       //----------------------------------------------------------------------
       // 1000 mbar switches (APS)
       //----------------------------------------------------------------------
       // delayed 1000 mbar furnace chamber
       //----------------------------------
       #iTime := S_ODT(   
                   T_NO:= "BM_VAC_TMR_APS_FCH",              // Timer
                   S   := "PDI".FCH_APS,                     // Start Condition
                   TV  := #DELAY_APS_FCH,                   // Time Setpoint
                   R   := NOT "PDI".FCH_APS,                 // Reset Condition
                   BI  => #BI_TMR_APS_FCH,                  // Current Time Value
                   Q   => "DV".APS_FCH_DELAYED);             // Output


       // delayed 1000 mbar gate
       //-----------------------
       #iTime := S_ODT(   
                   T_NO:= "BM_VAC_TMR_APS_GCH",            // Timer
                   S   := "PDI".GCH_APS,                   // Start Condition
                   TV  := #DELAY_APS_GCH,                 // Time Setpoint
                   R   := NOT "PDI".GCH_APS,               // Reset Condition
                   BI  => #BI_TMR_APS_GCH,                // Current Time Value
                   Q   => "DV".APS_GCH_DELAYED);           // Output

       // delayed 1000 mbar feeder
       //-------------------------
       #iTime := S_ODT(   
                   T_NO:= "BM_VAC_TMR_APS_FDR",            // Timer
                   S   := "PDI".FDR_APS,                   // Start Condition
                   TV  := #DELAY_APS_FDR,                 // Time Setpoint
                   R   := NOT "PDI".FDR_APS,               // Reset Condition
                   BI  => #BI_TMR_APS_FDR,                // Current Time Value
                   Q   => "DV".APS_FDR_DELAYED);           // Output

       // delayed 1000 mbar main filter
       //------------------------------
       #iTime := S_ODT(   
                   T_NO:= "BM_VAC_TMR_APS_FIL",            // Timer
                   S   := "PDI".FIL_APS,                   // Start Condition
                   TV  := #DELAY_APS_FIL,                 // Time Setpoint
                   R   := NOT "PDI".FIL_APS,               // Reset Condition
                   BI  => #BI_TMR_APS_FIL,                // Current Time Value
                   Q   => "DV".APS_FIL_DELAYED);           // Output

       // delayed 1000 mbar bypass filter
       //--------------------------------
       #iTime := S_ODT(   
                   T_NO:= "BM_VAC_TMR_APS_BY_FIL",            // Timer
                   S   := "PDI".FIL_2_APS,                   // Start Condition
                   TV  := #DELAY_APS_BY_FIL,                 // Time Setpoint
                   R   := NOT "PDI".FIL_2_APS,               // Reset Condition
                   BI  => #BI_TMR_APS_BY_FIL,                // Current Time Value
                   Q   => "DV".APS_BY_FIL_DELAYED);           // Output


       "LT".CGT_APS      := "DV".APS_GCH_DELAYED;
       "LT".CLF_APS      := "DV".APS_FCH_DELAYED;
       "LT".FDR_APS      := "DV".APS_FDR_DELAYED;
       "LT".FIL_APS      := "DV".APS_FIL_DELAYED;
       "LT".BY_FIL_APS   := "DV".APS_BY_FIL_DELAYED;

       //----------------------------------------------------------------------
       // Select and set output for gas flow 1+2
       //----------------------------------------------------------------------
       "P_BM_SET_GAS_FLW_MFC_1":P := "CM_INSELECT"(auto := ("APC".AUTOMATIC AND NOT "SY".CTL_GAS_FLOW_SMI) OR "DV".SI_FIL_FSH_SEQ_ON,
                                           track:= true,
                                           ac   := "AC".SET_GAS_1_FLW,
                                           kya  := "KYA".SET_GAS_1_FLW);


       "P_BM_SET_GAS_FLW_MFC_2":P := "CM_INSELECT"(auto := "APC".AUTOMATIC AND NOT "SY".CTL_GAS_FLOW_SMI,
                                           track:= true,
                                           ac   := "AC".SET_GAS_2_FLW,
                                           kya  := "KYA".SET_GAS_2_FLW);
       IF NOT "SY".SIM_ON THEN
           "DIS".ACT_GAS_1_FLW    := "P_BM_ACT_GAS_FLW_MFC_1":P;
           "DIS".ACT_GAS_2_FLW    := "P_BM_ACT_GAS_FLW_MFC_2":P;
       END_IF;

       "LT".V16_1_OPEN := ("DIS".ACT_GAS_1_FLW>0.0) AND ("PDO".V5 OR "PDO".V6);
       "LT".V16_2_OPEN := ("DIS".ACT_GAS_2_FLW>0.0) AND ("PDO".V5 OR "PDO".V6);

       //reset manual gas flow setpoint when inlet valves are not open
       //-------------------------------------------------------------
       IF NOT ("LT".V5_OPEN OR "LT".V6_OPEN)   THEN
           "KYA".SET_GAS_1_FLW   :=  0.0;
           "KYA".SET_GAS_2_FLW   :=  0.0;
       END_IF;

       //--------------------------------------------------------------------
       //Process pump P1
       //--------------------------------------------------------------------
       "CM_ITL_IO"(ADR := 1,
                 KYD_ON := ("KYD".P1_ON OR "DV".PWR_FAIL_P1_ON),
                 KYD_OFF:= "KYD".P1_OFF,
                 AUTO := "APC".AUTOMATIC OR "DV".SI_FIL_FSH_SEQ_ON,
                 DC_ON:= "DC".P1_ON,
                 CON1 := "PDI".EMO, 
                 CON2 := NOT "DV".MAIN_LINE_FAULT, 
                 CON3 := "DV".MAIN_SWITCH_ON,
                 CON4 := "PDI".P1_FLT,
                 CON5 := NOT #Flt_P1,
                 CON6 := NOT "FLT".P1_TMP_HIGH,
                 CON7 := "SysLog1",
                 CON8 := "SysLog1",
                 ITL_OUT:= "STA_ITL_CAUSE",
                 LT_OUT := "LT".P1_ON);

       //delay P1 start
       //--------------
       "PDO".P1_ON   := "SysOndelay"( DIN := "LT".P1_ON,
                               SetTime := 10,                              // setp. time
                               ActTime := #p1_on_dly,                       // act. time
                               Tick    := "SysTick100ms");                   // timebase (1s)

       #P1_IS_ON := "PDO".P1_ON AND NOT "PDI".P1_IS_ON;             //PDI.P1_IS_ON = false: pump is running; true: pump is off

       #P1_NOT_READY := "SysOndelay"( DIN := "PDO".P1_ON AND "PDI".P1_IS_ON,
                               SetTime := 3,                           // setp. time
                               ActTime := #FltTimeP1,                   // act. time
                               Tick    := "SysTick1s");                  // timebase (1s)

       IF ("PDO".P1_ON AND #P1_NOT_READY) THEN
           #Flt_P1 := true;
       END_IF;
       (*
       //motor temperature monitoring of pump P1
       //---------------------------------------
       FLT.P1_TMP_HIGH := SysOndelay(  DIN     := NOT PDI.MON_TMP_P1,
                                       SetTime := 5,                           // setp. time
                                       ActTime := tmp_flt_p1_dly,              // act. time
                                       Tick    := SysTick1s);                  // timebase (1s)
       *)
       //reset of PTC tripping devices pump 1 and pump 2
       //-----------------------------------------------
       "LT".RST_SIHI_PU  := "SysOffdelay"( DIN     := "KYD".RST_SIHI_PU,          // reset button HMI
                                       SetTime := 10,                      // setp. time
                                       ActTime := #tmp_flt_p1_dly,          // act. time
                                       Tick    := "SysTick100ms");

       "PDO".MON_TMP_P2_RES :=  "LT".RST_SIHI_PU;     //output used for both pumps - P1 and P2                                

       //Read out SPGuard
       //-------------------------------------
       #Dprd_P1_RetVal  :=  DPRD_DAT(   LADDR  :=  16#400,             //addr1024 
                                        RECORD =>  #P1_DATA); 

       "DIS".ACT_VIB_P1          := (BYTE_TO_INT(#P1_DATA[1])-48)* 1000.0 + (BYTE_TO_INT(#P1_DATA[2])-48)*100.0 + 
                                  (BYTE_TO_INT(#P1_DATA[3])-48)*10.0 + (BYTE_TO_INT(#P1_DATA[4])-48)*1.0;
       "DIS".ACT_GEAR_OIL_TMP_P1 := (BYTE_TO_INT(#P1_DATA[6])-48)*10.0 + (BYTE_TO_INT(#P1_DATA[7])-48)* 1.0;

       "FLT".P1 := #Flt_P1 OR NOT "PDI".P1_FLT;    
       "FLT".MSR_P1_VIB           := "DIS".ACT_VIB_P1 > 149.0;
       "FLT".P1_GEAR_OIL_TMP_WRN  := "DIS".ACT_GEAR_OIL_TMP_P1> 60.0;
       "FLT".P1_GEAR_OIL_TMP_ALM  := "DIS".ACT_GEAR_OIL_TMP_P1>70.0;
       "FLT".P1_SP_WRN            := "PDI".P1_WRN OR (#P1_DATA[8]=B#16#31); 

       //--------------------------------------------------------------------
       //V10 SECUVAC Ventil P1
       //--------------------------------------------------------------------
       "PDO".V10 := "PDO".P1_ON;

       //----------------------------------------------------------------------
       // V9_1 open/close : Vacuum pump 1 seal gas         
       //----------------------------------------------------------------------
       (*
       V9_1_dly_op := SysOndelay(  DIN     := PDO.P1_ON,
                                   SetTime := 10,                      // setp. time
                                   ActTime := DelayV9_1,               // act. time
                                   Tick    := SysTick1s);              // timebase (1s)
       *)                            
       //seal gas valve vacuum pump 1 - valve opened before pump starts
       //--------------------------------------------------------------
       "PDO".P1_SEAL_GAS :=  "SysOffdelay"(DIN     := "PDI".EMO AND "DV".MAIN_SWITCH_ON AND "LT".P1_ON,
                                       SetTime := 3600,                        // setp. time
                                       ActTime := #p1_seal_gas_off_dly,         // act. time
                                       Tick    := "SysTick1s");                  // timebase (1s)
       (*
       //gas ballast valve vacuum pump 1
       //-------------------------------
       PDO.P1_GAS_BAL :=       PDI.EMO 
                           AND DV.MAIN_SWITCH_ON 
                           AND PDO.P1_ON
                           AND DV.P1_GAS_BAL_ENB;
       *)
       //--------------------------------------------------------------------
       //Booster pump P2
       //--------------------------------------------------------------------
       "PDO".P2_ON := "PDO".P1_ON AND NOT "FLT".P2_TMP_HIGH;
       "PDO".P2_FU_ON := "PDO".P1_ON AND #V2_ONDELAY_OVER;

       #P2_NOT_READY := "SysOndelay"( DIN := "PDO".P2_FU_ON AND NOT "PDI".FU_P2_RDY,
                               SetTime := 5,                           // setp. time
                               ActTime := #FltTimeP2,                   // act. time
                               Tick    := "SysTick1s");                  // timebase (1s)

       IF ("PDO".P2_FU_ON AND #P2_NOT_READY) THEN
           #Flt_P2 := true;
       ELSE
           #Flt_P2 := false;
       END_IF;

       "FLT".P2 := #Flt_P2;

       "PDO".P2_FU_RES := "KYD".ALARM_ACKN AND NOT #P2_NOT_READY;   

       //motor temperature monitoring of pump P2
       //---------------------------------------
       "FLT".P2_TMP_HIGH := "SysOndelay"(  DIN     := "PDI".MON_TMP_P2,
                                       SetTime := 5,                           // setp. time
                                       ActTime := #tmp_flt_p2_dly,              // act. time
                                       Tick    := "SysTick1s");                  // timebase (1s)

       //--------------------------------------------------------------------
       //Process pump P3
       //--------------------------------------------------------------------
       #mob_fdr_p3_off_req  :=  #mob_fdr_p3_on_req AND NOT "DV".MOB_FDR_P3_ON_REQ;
       #mob_fdr_p3_on_req   :=  "DV".MOB_FDR_P3_ON_REQ;

       "CM_ITL_IO"(ADR := 2,
                 KYD_ON := ("KYD".P3_ON OR "DV".PWR_FAIL_P3_ON OR "DV".MOB_FDR_P3_ON_REQ),
                 KYD_OFF:= ("KYD".P3_OFF OR #mob_fdr_p3_off_req),
                 AUTO := "APC".AUTOMATIC OR "DV".FIL_CLN_REQ_IN_PRC,
                 DC_ON:= ("DC".P3_ON OR "DV".MOB_FDR_P3_ON_REQ OR "DV".P3_ON),
                 CON1 := "PDI".EMO, 
                 CON2 := NOT "DV".MAIN_LINE_FAULT, 
                 CON3 := "DV".MAIN_SWITCH_ON,
                 CON4 := NOT #Flt_P3,
                 CON5 := "SysLog1",
                 CON6 := "SysLog1",
                 CON7 := "SysLog1",
                 CON8 := "SysLog1",
                 ITL_OUT:= "STA_ITL_CAUSE",
                 LT_OUT := "PDO".P3_ON);

       "LT".P3_ON := "PDO".P3_ON;
       #P3_IS_ON := "PDO".P3_ON;

       IF ("PDO".P3_ON AND #P3_NOT_READY) THEN
           #Flt_P3 := true;
       END_IF;
       "FLT".P3 := #Flt_P3;


       // main line is on again
       //----------------------------------------------
       IF NOT "DV".MAIN_LINE_FAULT THEN  
               "DV".PWR_FAIL_P1_ON := false;
               "DV".PWR_FAIL_P3_ON := false;
       END_IF;

       // Reset fault message
       //----------------------------------------------
       IF "DV".ALARM_ACKN THEN
           #Flt_P1 := false;
           "FLT".P2 := false;
           #Flt_P3 := false;
       END_IF;



       //----------------------------------------------------------------------
       // Release V2 xx seconds after P1 on
       //----------------------------------------------------------------------
       #iTime := S_ODT(
                   T_NO:= "BM_VAC_TMR_V2_ON",            // Timer
                   S   := #P1_IS_ON,                    // Start Condition
                   TV  := #DELAY_TIME_V2_ON,            // Time Setpoint
                   R   := NOT #P1_IS_ON,                // Reset Condition
                   BI  => #BI_TMR_V2_ONDEL,             // Current Time Value
                   Q   => #V2_ONDELAY_OVER);            // Output

       //----------------------------------------------------------------------
       // open V3 xx seconds after P3 on
       //----------------------------------------------------------------------

       #iTime := S_ODT(
                   T_NO:= "BM_VAC_TMR_V3_ON",            // Timer
                   S   := #P3_IS_ON,                    // Start Condition
                   TV  := #DELAY_TIME_V3_ON,            // Time Setpoint
                   R   := NOT #P3_IS_ON,                // Reset Condition
                   BI  => #BI_TMR_V3_ONDEL,             // Current Time Value
                   Q   => #V3_ONDELAY_OVER);            // Output

       //----------------------------------------------------------------------
       // V 1: throttle valve position with softpumping
       //----------------------------------------------------------------------
       IF "DV".V1_HAND_MODE THEN //V1 hand mode from filter cleaning sequence during process is active
           #TRV_SET_POS :=  "KYA".SET_CTL_VALVE_POS;
       ELSE
           #TRV_SET_POS :=  "CTL".SET_CTL_VALVE_POS;
       END_IF;

       //built set point of pressure control valve V1
       //--------------------------------------------
       IF #V2_ONDELAY_OVER AND (("DV".ACC_ENB_VAC AND NOT "DV".FIL_VNT_REQ) OR "LT".SI_FIL_FSH_SEQ_ON)  THEN        //P1 on 
          IF ("PAR_MAIN".PD_SOFTPUMP_DELAY < 1.0) OR "SY".CTL_PRS_ON THEN 
             "PAO".TRV_SET_POS := #TRV_SET_POS;
          ELSE 
             #TRV_POS_INC := 10.0 / "PAR_MAIN".PD_SOFTPUMP_DELAY;  // 100 ms steps
             IF "SysTick100ms" THEN                // calculate in 100 ms steps
                IF "PAO".TRV_SET_POS < #TRV_SET_POS THEN
                   "PAO".TRV_SET_POS := "PAO".TRV_SET_POS + #TRV_POS_INC; 
                      IF "PAO".TRV_SET_POS > #TRV_SET_POS THEN
                         "PAO".TRV_SET_POS := #TRV_SET_POS;
                      END_IF;
                ELSE
                   "PAO".TRV_SET_POS := #TRV_SET_POS;
                END_IF;
             END_IF;
          END_IF;
       ELSE
          "PAO".TRV_SET_POS := 0.0;
       END_IF;

       "PDO".V1_CL :=  ("PAO".TRV_SET_POS = 0.0); // V1 close exact when setpoint position is 0 

       "LT".V1_OPEN := ("PAI".TRV_ACT_POS >= 0.5);

       //write set point and actual value to display variables
       //-----------------------------------------------------
       IF "PDI".LS_V1_CL THEN 
          "DIS".ACT_CTL_VALVE_POS := 0.0;
       ELSE     
          "DIS".ACT_CTL_VALVE_POS := "PAI".TRV_ACT_POS;  
       END_IF;

       "DIS".SET_CTL_VALVE_POS   :=  "KYA".SET_CTL_VALVE_POS;

       // V 1.1: throttle valve for bypass filter
       //----------------------------------------
       //pump is off
       //-----------
       IF NOT #P1_IS_ON THEN
           #TRV_SET_POS_V1_1            :=  0.0;                //write manual set point
           "KYA".SET_CTL_VALVE_POS_V1_1  :=  #TRV_SET_POS_V1_1;   //track manual set point of pressure control valve V1.1
       //follow set point of V1 in pump down phase
       //-----------------------------------------
       ELSIF ("APC".STATUS = "APC".PUMP_DOWN) THEN
           IF "SysTick100ms" THEN
               IF "DC".V1_1_REL THEN         //release bit set in pump down phase
                   IF #TRV_SET_POS_V1_1 < "PAO".TRV_SET_POS THEN  //write set point of V1 to V1.1
                       #TRV_SET_POS_V1_1    :=  #TRV_SET_POS_V1_1 + #TRV_POS_INC; 
                   ELSE
                       #TRV_SET_POS_V1_1    :=  "PAO".TRV_SET_POS;
                   END_IF;
               END_IF;
           END_IF;
           "KYA".SET_CTL_VALVE_POS_V1_1  :=  #TRV_SET_POS_V1_1;   //track manual set point of pressure control valve V1.1
       //all other phases - use KYA value as set point which is only set in FB BM_FIL_CHG
       //--------------------------------------------------------------------------------
       ELSIF "DV".V1_1_HAND_MODE THEN
           #TRV_SET_POS_V1_1    :=  "KYA".SET_CTL_VALVE_POS_V1_1; //write manual set point
       //filter cleaning while process is running is active
       //--------------------------------------------------
       ELSE  
           #TRV_SET_POS_V1_1            :=  "CTL".SET_CTL_VALVE_POS;      //write controller output as set point
           "KYA".SET_CTL_VALVE_POS_V1_1  :=  #TRV_SET_POS_V1_1;           //track manual set point of pressure control valve V1.1
       END_IF;

       //set light variable
       //------------------
       "LT".V1_1_OPEN := ("PAI".TRV_ACT_POS_1 >= 0.5);

       //write set point to peripherie output
       //------------------------------------
       "PAO".TRV_SET_POS_1 := #TRV_SET_POS_V1_1;

       //set totallay close output of control valve
       //------------------------------------------
       "PDO".V1_1_CL :=  ("PAO".TRV_SET_POS_1 = 0.0);

       //write set point and actual value to display variables
       //-----------------------------------------------------
       "DIS".ACT_CTL_VALVE_POS_V1_1  :=  "PAI".TRV_ACT_POS_1;  
       "DIS".SET_CTL_VALVE_POS_V1_1  :=  #TRV_SET_POS_V1_1;

       //-----------------------------------------------
       // release gas valves after power fail
       //-----------------------------------------------
       IF "PDO".V2_1 THEN        
          "DV".V5_CLOSE_REQ := false;         // release gas valves v5 and v6
          "DV".V6_CLOSE_REQ := false;         // after power fail if v2.x open
       END_IF; 

       //----------------------------------------------------------------------
       // V 2.1 open/close  (Vacuum valve furnace chamber)
       //----------------------------------------------------------------------
       IF ("DV".SI_FIL_FSH_SEQ_ON OR "DV".V2_1_CL) THEN
          "PDO".V2_1  :=  FALSE;
       ELSIF (#P1_IS_ON AND ("LT".V1_OPEN OR "DV".FIL_CLN_REQ_IN_PRC)) THEN 
          "PDO".V2_1  :=  TRUE;
       END_IF;

       "LT".V2_1_OPEN := "PDI".LS_V2_1_OP;

       "FLT".V2_1 := "SysOndelay"(DIN := "PDO".V2_1 AND NOT "PDI".LS_V2_1_OP,
                              SetTime:= 5,                              // setp. time
                              ActTime := #FltTimeV2_1,                   // act. time
                              Tick:= "SysTick1s" );                       // timebase (1s)

       // V 2.11 open/close  (Bypass vacuum valve furnace chamber)
       //---------------------------------------------------------
       IF (("STA".ACT_DVC_CNF_BYTE_3 AND 2#1000_0000) = 2#1000_0000) THEN   
           //pump down phase - open V2.11 initially
           //--------------------------------------
           IF ("APC".STATUS = "APC".PUMP_DOWN) THEN
               //furnace pressure must be below 95 mbar - inside measurement range of gauge
               //--------------------------------------------------------------------------
               IF ("DIS".ACT_PRS_CLF < 95.0) THEN
                   IF "LT".V1_1_OPEN AND ("DIS".ACT_PRS_BYP_FIL < 1.0) THEN    //bypass filter pressure must be below 1 mbar
                       "PDO".V2_11  :=  TRUE;
                   END_IF;
               END_IF;
           //all other phases - use DV value as opening trigger which is only set in FB BM_FIL_CHG
           //-------------------------------------------------------------------------------------
           ELSIF (#P1_IS_ON AND "DV".V2_11_OP) THEN     
               "PDO".V2_11  :=  TRUE;
           //close valve outside pump down phase and filter cleaning sequence
           //----------------------------------------------------------------
           ELSE
               "PDO".V2_11  :=  FALSE;
           END_IF;

           "LT".V2_11_OPEN := "PDI".LS_V2_11_OP;

           //set valve position alarm
           //------------------------
           "FLT".V2_11 := "SysOndelay"(DIN := "PDO".V2_11 AND NOT "PDI".LS_V2_11_OP,
                                   SetTime:= 5,                                // setp. time
                                   ActTime := #FltTimeV2_11,                    // act. time
                                   Tick:= "SysTick1s" );                         // timebase (1s)
       END_IF;

       IF (("STA".ACT_DVC_CNF_BYTE_3 AND 2#0010_0000) = 2#0010_0000) THEN        //nur f黵 Test, l鰏chen wenn Ventil ausgebaut ist
           "PDO".V2_11  :=  TRUE;
       END_IF;

         //----------------------------------------------------------------------
         // V 3 open/close (Vacuum valve gate chamber)
         //----------------------------------------------------------------------
          "CM_ITL_IO"(ADR := 5,
                 KYD_ON := "KYD".V3_OPEN,
                 KYD_OFF:= "KYD".V3_CLOSE,
                 AUTO := "APC".AUTOMATIC,
                 DC_ON:= "DC".V3_OP,
                 CON1 := "PDI".EMO, 
                 CON2 := "DV".MAIN_SWITCH_ON, 
                 CON3 := #P3_IS_ON,
                 CON4 := #V3_ONDELAY_OVER,                          // P3 is on
                 CON5 := NOT "PDO".V3_2,                             // vacuum valve feeder closed
                 CON6 := NOT "PDO".V4,
                 CON7 := ("PDI".LS_V7_SW_IN AND "PDI".LS_V7_DN),    // Gate valve closed
                 CON8 := "SysLog1",
                 ITL_OUT:= "STA_ITL_CAUSE",
                 LT_OUT := "PDO".V3);

          "LT".V3_OPEN  := "PDI".LS_V3_OP;

          "FLT".V3   := "SysOndelay"( DIN := "PDO".V3 AND NOT "PDI".LS_V3_OP,
                                  SetTime:= 5,                              // setp. time
                                  ActTime := #FltTimeV3,                     // act. time
                                  Tick:= "SysTick1s");                    // timebase (1s)

         //----------------------------------------------------------------------
         // V 3.2 open/close (vacuum valve feeder)
         //----------------------------------------------------------------------
          #mob_fdr_v3_2_cl_req    :=  #mob_fdr_v3_2_opn_req AND NOT "DV".MOB_FDR_V3_2_OPN_REQ;
          #mob_fdr_v3_2_opn_req   :=  "DV".MOB_FDR_V3_2_OPN_REQ;

          "CM_ITL_IO"(ADR := 6,
                 KYD_ON := ("KYD".V3_2_OP OR "DV".MOB_FDR_V3_2_OPN_REQ),
                 KYD_OFF:= ("KYD".V3_2_CL OR #mob_fdr_v3_2_cl_req),
                 AUTO := "APC".AUTOMATIC,
                 DC_ON:= ("DC".V3_2_OP OR "DV".MOB_FDR_V3_2_OPN_REQ),
                 CON1 := "PDI".EMO, 
                 CON2 := "DV".MAIN_SWITCH_ON, 
                 CON3 := #P3_IS_ON,
                 CON4 := #V3_ONDELAY_OVER,                          // P3 is on
                 CON5 := NOT "PDO".V3,                               // vacuum valve gate chamber closed
                 CON6 := ("PDI".LS_V11_CL AND NOT "PDI".LS_V11_OP),    // isolation valve feeder closed,
                 CON7 := NOT "PDO".V24,                              // valve argon inlet feeder closed 
                 CON8 := "DV".MOB_FDR_V11_INST,                      // mobile feeder valve installed
                 ITL_OUT:= "STA_ITL_CAUSE",
                 LT_OUT := "PDO".V3_2);

          "LT".V3_2_OP  := "PDO".V3_2;




       //----------------------------------------------------------------------
       // V 3.3 open/close (main filter)
       //----------------------------------------------------------------------
       "CM_ITL_IO"(ADR := 14,
                 KYD_ON    := "KYD".V3_3_OP,
                 KYD_OFF   := "KYD".V3_3_CL,
                 AUTO      := "APC".AUTOMATIC OR "DV".FIL_CLN_REQ_IN_PRC,
                 DC_ON     := "DV".V3_3_OP,
                 CON1      := "PDI".EMO, 
                 CON2      := "DV".MAIN_SWITCH_ON, 
                 CON3      := #V3_ONDELAY_OVER,                      //valve open delay is over
                 CON4      := NOT "PDO".V3,                           //vacuum valve to gate closed
                 CON5      := NOT "PDO".V3_2,                         //vacuum valve feeder closed
                 CON6      := NOT "PDO".V4,                           //Ar vent valve is closed
                 CON7      := NOT "PDO".V3_4,                         //vacuum valve to bypass filter closed
                 CON8      := "SysLog1",
                 ITL_OUT   := "STA_ITL_CAUSE",
                 LT_OUT    := "PDO".V3_3);

       "LT".V3_3_OPEN  := "PDI".LS_V3_3_OP;

       "FLT".V3_3   := "SysOndelay"( DIN := "PDO".V3_3 AND NOT "PDI".LS_V3_3_OP,
                                  SetTime:= 5,                             // setp. time
                                  ActTime := #FltTimeV3_3,                  // act. time
                                  Tick:= "SysTick1s");                       // timebase (1s)

       //----------------------------------------------------------------------
       // V 3.4 open/close (bypass filter)
       //----------------------------------------------------------------------
       "CM_ITL_IO"(ADR := 15,
                 KYD_ON    := "KYD".V3_4_OP,
                 KYD_OFF   := "KYD".V3_4_CL,
                 AUTO      := "APC".AUTOMATIC OR "DV".FIL_CLN_REQ_IN_PRC,
                 DC_ON     := "DC".V3_4_OP OR "DV".V3_4_OP,
                 CON1      := "PDI".EMO, 
                 CON2      := "DV".MAIN_SWITCH_ON, 
                 CON3      := #V3_ONDELAY_OVER,                      //valve open delay is over
                 CON4      := NOT "PDO".V3,                           //vacuum valve to gate closed
                 CON5      := NOT "PDO".V3_2,                         //vacuum valve feeder closed
                 CON6      := NOT "PDO".V4,                           //Ar vent valve is closed
                 CON7      := NOT "PDO".V3_3,                         //vacuum valve to main filter closed
                 CON8      := "SysLog1",
                 ITL_OUT   := "STA_ITL_CAUSE",
                 LT_OUT    := "PDO".V3_4);

          "LT".V3_4_OPEN  := "PDI".LS_V3_4_OP;

          "FLT".V3_4   := "SysOndelay"( DIN := "PDO".V3_4 AND NOT "PDI".LS_V3_4_OP,
                                  SetTime:= 5,                             // setp. time
                                  ActTime := #FltTimeV3_4,                  // act. time
                                  Tick:= "SysTick1s");                       // timebase (1s)

         //----------------------------------------------------------------------
         // V 4 open/close  (Gas inlet valve gate chamber)
         //----------------------------------------------------------------------
         IF "LT".ACC_OVP_TEST_ON THEN
            "PDO".V4 :=   "PDI".EMO AND "DV".ACC_OVP_TEST_ON;  //open V4 when over pressure test is active - bypass interlocks  
         ELSE
          "CM_ITL_IO"(ADR := 7,
                 KYD_ON := "KYD".V4_OPEN ,
                 KYD_OFF:= "KYD".V4_CLOSE,
                 AUTO := "APC".AUTOMATIC OR "DV".SI_FIL_FSH_SEQ_ON,
                 DC_ON:= "DC".V4_OP,
                 CON1 := "PDI".EMO, 
                 CON2 := "DV".MAIN_SWITCH_ON,
                 CON3 := NOT "DV".APS_GCH_DELAYED, 
                 CON4 := (NOT "LT".V1_OPEN OR ("PDI".LS_V7_SW_IN AND "PDI".LS_V7_DN)),
                 CON5 := "DV".ACC_ENB_GAS_V,  
                 CON6 := "SysLog1",                     
                 CON7 := "SysLog1",    
                 CON8 := "SysLog1",   
                 ITL_OUT:= "STA_ITL_CAUSE",
                 LT_OUT := "PDO".V4);
         END_IF;
          "LT".V4_OPEN  := "PDO".V4;


         //----------------------------------------------------------------------
         //set auto open flag of valve V6
         //--------------------------------------------------------------
          IF  "PDO".V5                                                                                AND NOT 
              "PDI".LS_V7_SW_OUT                                                                      AND
              (("KYA".SET_GAS_1_FLW > 0.1) OR ("KYA".SET_GAS_2_FLW > 0.1))                              AND 
              ("LT".HTR_1_ON OR "LT".HTR_2_ON OR ("AV".ACT_HTR_1_TMP >= "CNF".HTR_1_TMP_RANGE_LOW + 50.0))  THEN

              #v6_auto_opn_req    :=  TRUE;
              #v5_auto_cl_req     :=  "PDI".LS_V7_SW_IN AND "PDI".LS_V7_DN;
          ELSE
              #v6_auto_opn_req    :=  FALSE;
              #v5_auto_cl_req     :=  FALSE;
          END_IF;

          //set auto close flag of valve V6 
          //--------------------------------------------------------------
          IF   "PDO".V6                                                                                AND  
              (("KYA".SET_GAS_1_FLW > 0.1) OR ("KYA".SET_GAS_2_FLW > 0.1))                               AND 
              ("LT".HTR_1_ON OR "LT".HTR_2_ON OR ("AV".ACT_HTR_1_TMP >= "CNF".HTR_1_TMP_RANGE_LOW + 50.0))   THEN

              #v6_auto_cl_req    := "PDI".LS_V7_SW_OUT AND "PDI".LS_V7_UP;
              #v5_auto_opn_req   := "PDI".LS_V7_UP AND NOT "PDI".LS_V7_SW_IN AND NOT "PDO".V5; 

          ELSE
              #v6_auto_cl_req    :=  FALSE;
              #v5_auto_opn_req   :=  FALSE;
          END_IF;

          //delay auto close flag of valve V6
          //---------------------------------
          IF #v6_auto_cl_req OR #v6_cl_dly_run THEN 
              #v6_cl_dly_run   :=  true;     
              IF (#i < 5) THEN
                  IF "SysTick100ms" THEN
                      #i := #i + 1;
                  END_IF;
              ELSE
                  #v6_auto_cl_req_dly  :=  true;
                  #v6_cl_dly_run       :=  false;
              END_IF;
          ELSE
              #v6_auto_cl_req_dly  :=  false;
              #i                   :=  0;
          END_IF;

         //store status of gate valve closed LS in the running cycle
         //---------------------------------------------------------    
         #cgt_v_cld_prv   :=  "PDI".LS_V7_SW_IN AND "PDI".LS_V7_DN;

         //----------------------------------------------------------------------
         // V 5 open/close   (Controlled gas inlet valve gate chamber)
         //----------------------------------------------------------------------
          "CM_ITL_IO"(ADR := 8,
                 KYD_ON := ("KYD".V5_OPEN OR #v5_auto_opn_req),
                 KYD_OFF:= ("KYD".V5_CLOSE OR #v5_auto_cl_req OR "DV".V5_CLOSE_REQ),
                 AUTO := "APC".AUTOMATIC,
                 DC_ON:= "DC".V5_OP,
                 CON1 := "PDI".EMO,
                 CON2 := "DV".MAIN_SWITCH_ON,
                 CON3 := NOT "DV".APS_GCH_DELAYED, 
                 CON4 := NOT ("PDI".LS_V7_SW_IN AND "PDI".LS_V7_DN),                 //close V5 if gate valve is closed  
                 CON5 := "DV".ACC_ENB_GAS_V,   
                 CON6 := "SysLog1",                     
                 CON7 := "SysLog1",    
                 CON8 := "SysLog1",   
                 ITL_OUT:= "STA_ITL_CAUSE",
                 LT_OUT := "PDO".V5);

          "LT".V5_OPEN  := "PDO".V5;

         //----------------------------------------------------------------------
         // V 6 open/close   (Controlled gas inlet valve furnace chamber)
         //----------------------------------------------------------------------
          "CM_ITL_IO"(ADR := 9,
                 KYD_ON := ("KYD".V6_OPEN OR #v6_auto_opn_req),
                 KYD_OFF:= ("KYD".V6_CLOSE OR #v6_auto_cl_req_dly OR "DV".V6_CLOSE_REQ),
                 AUTO := "APC".AUTOMATIC OR "DV".SI_FIL_FSH_SEQ_ON,
                 DC_ON:= ("DC".V6_OP OR ("DC".V5_OP AND NOT "PDI".LS_V7_SW_OUT)),  //open V6 if gate valve is close,
                 CON1 := "PDI".EMO,
                 CON2 := "DV".MAIN_SWITCH_ON,
                 CON3 := NOT "DV".APS_FCH_DELAYED, 
                 CON4 := "DV".ACC_ENB_GAS_V,   
                 CON5 := "SysLog1",   
                 CON6 := "SysLog1",                     
                 CON7 := "SysLog1",    
                 CON8 := "SysLog1",   
                 ITL_OUT:= "STA_ITL_CAUSE",
                 LT_OUT := "PDO".V6);

          "LT".V6_OPEN  := "PDO".V6;

         //----------------------------------------------------------------------
         // V9.2 open/close (vent vacuum pipe gate pump side)
         //----------------------------------------------------------------------
         "DV".V9_2_DLY_OP := "SysOndelay"( DIN     := NOT "PDO".P3_ON,
                                       SetTime := 10,                      // setp. time
                                       ActTime := #DelayV9_2,               // act. time
                                       Tick    := "SysTick1s");              // timebase (1s)

         #V9_2_dly_cl := "SysOndelay"( DIN     := "DV".V9_2_DLY_OP,
                                    SetTime := 120,                     // setp. time
                                    ActTime := #onTimeV9_2,              // act. time
                                    Tick    := "SysTick1s");              // timebase (1s)


         "PDO".V9_2 :=   "PDI".EMO AND 
                       "DV".MAIN_SWITCH_ON AND  
                       "DV".V9_2_DLY_OP AND      //variable used for gate chamber lifting interlock
                       NOT #V9_2_dly_cl;

         //----------------------------------------------------------------------
         //V19 (dust outlet valve filter)
         //----------------------------------------------------------------------
          "CM_ITL_IO"(ADR := 10,
                 KYD_ON := "KYD".V19_OPEN,
                 KYD_OFF:= "KYD".V19_CLOSE,
                 AUTO := "APC".AUTOMATIC OR "DV".SI_FIL_FSH_SEQ_ON,
                 DC_ON:= "DC".V19_OP,
                 CON1 := "PDI".EMO,
                 CON2 := "DV".MAIN_SWITCH_ON,
                 CON3 := NOT "LT".V1_OPEN, 
                 CON4 := NOT "PDO".V2_1,   
                 CON5 := "SysLog1",   
                 CON6 := "SysLog1",                     
                 CON7 := "SysLog1",    
                 CON8 := "SysLog1",   
                 ITL_OUT:= "STA_ITL_CAUSE",
                 LT_OUT := "PDO".V19);

          "LT".V19_OPEN  := "PDO".V19;

       // V20 open/close (air inlet for oxidation dust filter)
       //----------------------------------------------------------------------
          "CM_ITL_IO"(ADR := 14,
                 KYD_ON := "KYD".V20_OPEN,
                 KYD_OFF:= "KYD".V20_CLOSE,
                 AUTO := "APC".AUTOMATIC OR "DV".SI_FIL_FSH_SEQ_ON,
                 DC_ON:= "DC".V20_OP,
                 CON1 := "PDI".EMO,
                 CON2 := "DV".MAIN_SWITCH_ON,
                 CON3 := NOT "LT".V22_OPEN,
                 CON4 := NOT "PDO".V2_1,                                                       // valve 2.1 is close,   
                 CON5 := NOT "LT".V1_OPEN,                                                     // valve V1 is open,               
                 CON6 := NOT "PDO".P1_ON,           
                 CON7 := "SysLog1",                                                  
                 CON8 := "SysLog1",
                 ITL_OUT:= "STA_ITL_CAUSE",
                 LT_OUT := "PDO".V20);

          "LT".V20_OPEN := "PDO".V20;

         //----------------------------------------------------------------------
         //V22 (argon inlet valve main filter)
         //----------------------------------------------------------------------
          "CM_ITL_IO"(ADR := 11,
                 KYD_ON := "KYD".V22_OPEN,
                 KYD_OFF:= "KYD".V22_CLOSE,
                 AUTO := "APC".AUTOMATIC OR "DV".SI_FIL_FSH_SEQ_ON OR "DV".FIL_CLN_REQ_IN_PRC,
                 DC_ON:= "DC".V22_OP OR "DV".V22_OP,
                 CON1 := "PDI".EMO,
                 CON2 := "DV".MAIN_SWITCH_ON,
                 CON3 := NOT "LT".V1_OPEN, 
                 CON4 := NOT "PDO".V2_1,   
                 CON5 := ("DIS".ACT_PRS_AR_VSL >= ("CNF".MIN_PRS_AR_VSL - #prs_hyst_ar_vsl)),   
                 CON6 := NOT "DV".APS_FIL_DELAYED,                     
                 CON7 := "SysLog1",    
                 CON8 := "SysLog1",   
                 ITL_OUT:= "STA_ITL_CAUSE",
                 LT_OUT := "PDO".V22);

           "LT".V22_OPEN:= "PDO".V22;

         //----------------------------------------------------------------------
         //V22.1 (argon inlet valve bypass filter)
         //----------------------------------------------------------------------
          "CM_ITL_IO"(ADR := 28,
                 KYD_ON := "KYD".V22_1_OP,
                 KYD_OFF:= "KYD".V22_1_CL,
                 AUTO := "APC".AUTOMATIC OR "DV".FIL_CLN_REQ_IN_PRC,
                 DC_ON:= "DV".V22_1_OP,
                 CON1 := "PDI".EMO,
                 CON2 := "DV".MAIN_SWITCH_ON,
                 CON3 := NOT "LT".V1_1_OPEN, 
                 CON4 := NOT "PDO".V2_11,   
                 CON5 := NOT "DV".APS_BY_FIL_DELAYED,   
                 CON6 := "SysLog1",                     
                 CON7 := "SysLog1",    
                 CON8 := "SysLog1",   
                 ITL_OUT:= "STA_ITL_CAUSE",
                 LT_OUT := "PDO".V22_1);

          "LT".V22_1_OPEN:= "PDO".V22_1;

         //----------------------------------------------------------------------
         // V24 open/close (argon inlet feeder)
         //----------------------------------------------------------------------
         #mob_fdr_v24_cl_req    :=  #mob_fdr_v24_opn_req AND NOT "DV".MOB_FDR_V24_OPN_REQ;
         #mob_fdr_v24_opn_req   :=  "DV".MOB_FDR_V24_OPN_REQ;

         "CM_ITL_IO"(ADR := 12,
                 KYD_ON := ("KYD".V24_OP OR "DV".MOB_FDR_V24_OPN_REQ),
                 KYD_OFF:= ("KYD".V24_CL OR #mob_fdr_v24_cl_req),
                 AUTO := "APC".AUTOMATIC,
                 DC_ON:= ("DC".V24_OP OR "DV".MOB_FDR_V24_OPN_REQ),
                 CON1 := "PDI".EMO,
                 CON2 := "DV".MAIN_SWITCH_ON,
                 CON3 := NOT "DV".APS_FDR_DELAYED, 
                 CON4 := "DV".MOB_FDR_V11_INST,   
                 CON5 := NOT "PDO".V3_2,                    //feeder vacuum valve is not open
                 CON6 := "SysLog1",                     
                 CON7 := "SysLog1",    
                 CON8 := "SysLog1",
                 ITL_OUT:= "STA_ITL_CAUSE",
                 LT_OUT := "PDO".V24);

          "LT".V24_OP  := "PDO".V24;

         //----------------------------------------------------------------------
         // V21 open/close (air inlet for oxidation process)
         //----------------------------------------------------------------------
          "CM_ITL_IO"(ADR := 13,
                 KYD_ON := "KYD".V21_OPEN,
                 KYD_OFF:= "KYD".V21_CLOSE,
                 AUTO := "APC".AUTOMATIC,
                 DC_ON:= "DC".V21_OP,
                 CON1 := "PDI".EMO,
                 CON2 := "DV".MAIN_SWITCH_ON,
                 CON3 := NOT "DV".APS_FCH_DELAYED,                                               // furnace pressure below 1000 mbar
                 CON4 :=(("PDO".V2_1 AND "PDI".LS_V2_1_OP AND                                      // valve 2.1 is open  
                         ("DIS".ACT_CTL_VALVE_POS > "CNF".REL_V21_POS_V1) AND                      // pressure control valve V1 is above 10% level
                         ("DIS".SET_CTL_VALVE_POS > "CNF".REL_V21_POS_V1))                         // set point is above 10 % level or
                         OR                       
                         (("PDO".V2_11 AND "PDI".LS_V2_11_OP OR (("STA".ACT_DVC_CNF_BYTE_3 AND 2#0010_0000) = 2#0010_0000)) //valve 2.11 is open or cooling tube without valve installed
                         AND 
                         ("DIS".ACT_CTL_VALVE_POS_V1_1 > "CNF".REL_V21_POS_V1) AND                 // pressure control valve V1.1 is above 10% level and  
                         ("DIS".SET_CTL_VALVE_POS_V1_1 > "CNF".REL_V21_POS_V1))),                  // set point is above 10 % level
                 CON5 := "SysLog1",
                 CON6 := (("DIS".ACT_GAS_1_FLW + "DIS".ACT_GAS_2_FLW) > 40.0),                     // gas flow 1 + 2 is > 40.0 l/min
                 CON7 := (("PDO".V5 AND "PDI".LS_V7_SW_OUT AND "PDI".LS_V7_UP) OR "PDO".V6),           // valve 5 and gate valve are open or valve 6 is open,                     
                 CON8 := #P1_IS_ON,                                                             // vacuum pump is running
                 ITL_OUT:= "STA_ITL_CAUSE",
                 LT_OUT := "PDO".V21);

          "LT".V21_OPEN := "PDO".V21;

          "FLT".V21_NOT_OPEN    :=  "SysOndelay"( DIN     := "APC".AUTOMATIC AND "DC".V21_OP AND NOT "PDO".V21,
                                              SetTime := 5,                       // setp. time
                                              ActTime := #v21_not_open_dly,        // act. time
                                              Tick    := "SysTick1s");              // timebase (1s)

         //----------------------------------------------------------------------
         // V25 open/close (argon inlet pressure storage tank)
         //----------------------------------------------------------------------
         "CM_ITL_IO"(ADR := 28,
                 KYD_ON := "KYD".V25_OPEN,
                 KYD_OFF:= "KYD".V25_CLOSE,
                 AUTO := "APC".AUTOMATIC OR "DV".SI_FIL_FSH_SEQ_ON OR "DV".FIL_CLN_REQ_IN_PRC,
                 DC_ON:= "DV".V25_OP,
                 CON1 := "PDI".EMO,
                 CON2 := "DV".MAIN_SWITCH_ON,
                 CON3 := NOT "PDO".V22, 
                 CON4 := ("DIS".ACT_PRS_AR_VSL <= ("CNF".MAX_PRS_AR_VSL + #prs_hyst_ar_vsl)),   
                 CON5 := "SysLog1",                    
                 CON6 := "SysLog1",                     
                 CON7 := "SysLog1",    
                 CON8 := "SysLog1",
                 ITL_OUT:= "STA_ITL_CAUSE",
                 LT_OUT := "PDO".V25);

          "LT".V25_OPEN := "PDO".V25;

        //-----------------------------V7------------------------
          "DV".LS_V7_SW_IN_DLY := "SysOndelay"( DIN := "PDI".LS_V7_SW_IN,
                                        SetTime:= 3,                             // setp. time
                                        ActTime := #TimeV7_SW_IN,                 // act. time
                                        Tick:= "SysTick1s"    );
          "DV".LS_V7_SW_OUT_DLY := "SysOndelay"( DIN := "PDI".LS_V7_SW_OUT,
                                        SetTime:= 3,                             // setp. time
                                        ActTime := #TimeV7_SW_OUT,                // act. time
                                        Tick:= "SysTick1s"    );
          "DV".LS_V7_UP_DLY  := "SysOndelay"( DIN := "PDI".LS_V7_UP,
                                        SetTime:= 3,                             // setp. time
                                        ActTime := #TimeV7_UP,                    // act. time
                                        Tick:= "SysTick1s"    );
          "DV".LS_V7_DN_DLY  := "SysOndelay"( DIN := "PDI".LS_V7_DN,
                                        SetTime:= 3,                             // setp. time
                                        ActTime := #TimeV7_DN,                    // act. time
                                        Tick:= "SysTick1s"    );       

          "FLT".V7   := "SysOndelay"( DIN := NOT (("PDI".LS_V7_SW_IN AND "PDI".LS_V7_DN) OR "PDI".LS_V7_SW_OUT AND "PDI".LS_V7_UP),
                                 SetTime:= 60,                             // setp. time
                                 ActTime := #FltTimeV7,                     // act. time
                                 Tick:= "SysTick1s"    );                    // timebase (1s)
END_FUNCTION_BLOCK

FUNCTION_BLOCK "BM_FIL_CHG"   // FB501, SCL
{ S7_Optimized_Access := 'FALSE' }
VERSION : 0.0
// -----------------------------------------------------------------------------------
//     program:         BM_FIL_CHG
//     description :    Filter change
//     name:            John Wang
//     date        :    11.02.2020
// 
//     revision    :   
//     name        :   
//     Date        :   
//     
//    
//     
//                     (c)PVA TePla AG
// -----------------------------------------------------------------------------------
   VAR
      flt_fil_chg : Bool;
      fil_cln_req_in_prc : Bool;
      fill_up_sto_tank : Bool;
      dly : Int;
      "step" : Int;
      i : Int;
      count : Int;
      fil_cln_off_dly : Int;
   END_VAR
   VAR_TEMP
      fil_chg_enb : Bool;
      k : Int;
   END_VAR
   VAR CONSTANT
      PRS_CTRL_V1_RMP : Real := 0.02;   // pressure control valve set point valve V1 ramp gradient
      PRS_CTRL_V1_1_RMP : Real := 0.02;   // pressure control valve set point valve V1.1 ramp gradient
      min_start_prs_by_fil : Real := 98.0;   // minimum pressure of bypass filter at sequence start [mbar]
   END_VAR
BEGIN


       #flt_fil_chg:= "FLT".V2_1 OR "FLT".V2_11 OR "FLT".V3_3; // OR FLT.V3_4;

       //write display values of main and bypass filter pressure
       //-------------------------------------------------------
       "DIS".ACT_PRS_MAIN_FIL    :=  "PAI".TRV_PRS_FIL_1;
     //DIS.ACT_PRS_BYP_FIL     :=  PAI.TRV_PRS_FIL_2;

       //pressure difference main filter to furnace chamber
       //--------------------------------------------------
       "DIS".PRS_DIFF_FIL_TO_FCH  :=  "PAI".TRV_PRS_FIL_1 - "PAI".FCH_BAR_ACT_PRS_100; 

       //write display value of argon tank pressure
       //------------------------------------------
       "DIS".ACT_PRS_AR_VSL      :=  "PAI".ACT_PRS_AR_VSL;

       //set enable bit filter cleaning during process
       //---------------------------------------------
       #fil_chg_enb :=      ("PAR_SUB".FIL_CHG_V1_POS >= 10.0)
                       AND NOT "PDI".P1_IS_ON                    //false: pump is running; true: pump is off
                       AND "SY".CTL_PRS_ON
                       AND NOT #flt_fil_chg;

       // set start bit main filter cleaning 
       //-----------------------------------
       IF (("DIS".SET_CTL_VALVE_POS >= "PAR_SUB".FIL_CHG_V1_POS) AND #fil_chg_enb AND "PDI".LS_V2_1_OP AND NOT #fil_cln_req_in_prc) THEN  
           //delay start after condition true
           //--------------------------------              
           IF (#dly > 60) THEN
               #fil_cln_req_in_prc := TRUE ;
           ELSE 
               IF "SysTick1s" THEN 
                   #dly   :=  #dly + 1;
               END_IF;
           END_IF;
       ELSE
           #dly :=  0;              //reset always when condition is not true
       END_IF;

       //stop sequence when automatic is switched off during abort sequence
       //------------------------------------------------------------------
       IF ("LT".ABORT_FIL_CLN AND NOT "APC".AUTOMATIC) THEN 
           #fil_cln_req_in_prc := FALSE;
       END_IF;

       //fill up gas storage tank
       //------------------------
       IF #fill_up_sto_tank THEN
           IF ("DIS".ACT_PRS_AR_VSL < "CNF".MAX_PRS_AR_VSL) THEN
               //open valve V25
               //--------------
               "DV".V25_OP   :=  TRUE;
           ELSE
               //close valve V25
               //--------------
               "DV".V25_OP           :=  FALSE;
               #fill_up_sto_tank    :=  false;  //fill up finished
           END_IF;
       END_IF;

       //sequence filter cleaning during process
       //---------------------------------------
       IF #fil_cln_req_in_prc THEN 
           //abort filter cleaning manually
           //------------------------------
           IF ("KYD".ABORT_FIL_CLN AND NOT "LT".ABORT_FIL_CLN) THEN
               #step                :=  2000;
               "LT".ABORT_FIL_CLN    :=  TRUE;
           END_IF;

           //filter change steps
           //-------------------
           CASE #step OF 

                 0://initialisation step
                   //-------------------
                   #count                   :=  0;
                   #i                       :=  0;
                   #fill_up_sto_tank        :=  true;                                           //request fill up of storage tank
                   IF (("STA".ACT_DVC_CNF_BYTE_3 AND 2#0010_0000) = 2#0010_0000) THEN
                       #step                :=  #step + 300;     //without bypass filter
                   ELSE                
                       #step                :=  #step + 50;      //with bypass filter
                   END_IF;
                   "LT".SI_FIL_FSH_SEQ_ON    :=  TRUE;
                   "DV".P3_ON                :=  TRUE;

                50://check if bypass filter pressure is above minimum start value
                   //------------------------------------------------------------
                   IF ("DIS".ACT_PRS_BYP_FIL < #min_start_prs_by_fil) THEN
                       "DV".V22_1_OP         := TRUE;
                   ELSE
                       //increase step counter
                       //---------------------
                       IF "SysTick1s" THEN
                           #i   :=  #i + 1;
                       END_IF;

                       //close valve V22.1
                       //-----------------
                       IF (#i >= 3) THEN    
                           "DV".V22_1_OP := FALSE;

                           //switch to next step
                           //-------------------
                           IF (#i > 3) THEN    
                               #step    :=  #step + 50;
                               #i       := 0;
                           END_IF;

                       END_IF;
                   END_IF;

               100://open V3.4 after delay when P3 is running
                   //----------------------------------------
                   IF "LT".P3_ON THEN 
                       IF "SysTick1s" THEN
                           #i   :=  #i + 1;
                       END_IF;
                       //increase step counter
                       //---------------------
                       IF (#i > 60) THEN    
                           "DV".V3_4_OP  :=  TRUE;
                           IF "PDI".LS_V3_4_OP THEN    
                               #step        :=  #step + 100;
                               #i           :=  0;
                           END_IF;
                      END_IF;
                   END_IF;

               200://if bypass filter pressure reached furnace chamber pressure then close V3.4 and wait 1s open v2.11
                   //-------------------------------------------------------------------------------------------------
                   IF ("DIS".ACT_PRS_CLF >= "DIS".ACT_PRS_BYP_FIL) THEN
                       "DV".V3_4_OP  := FALSE;
                       IF "PDI".LS_V3_4_CL THEN 
                           IF "SysTick100ms" THEN
                               #i   :=  #i + 1;
                           END_IF;
                           IF (#i > 10) THEN 
                               "DV".V2_11_OP := TRUE;
                               #step        :=  #step + 100;
                               #i           :=  0;
                           END_IF;
                       END_IF;
                   END_IF;

               300://hold set point of valve V1 
                   //--------------------------
                   IF ("PDI".LS_V2_11_OP OR (("STA".ACT_DVC_CNF_BYTE_3 AND 2#0010_0000) = 2#0010_0000)) THEN
                       "DV".V1_HAND_MODE:= TRUE;
                       //switch to next step
                       //-------------------
                       IF (#i > 10) THEN 
                           #step    :=  #step + 100;
                           #i       :=  0;
                       ELSIF "SysTick100ms" THEN
                           #i   :=  #i + 1;
                       END_IF;
                   END_IF; 

               400://reset pressure controller output
                   //--------------------------------
                   //switch to next step
                   //-------------------
                   IF (#i > 10) THEN 
                       #step    :=  #step + 100;
                       #i       :=  0;
                   ELSIF "SysTick100ms" THEN
                       "KYD".PRS_CTRL_RST    :=  TRUE;
                       #i   :=  #i + 1;
                   END_IF;

               500://transfer pressure control output to set point of V1.1
                   //-----------------------------------------------------
                   "KYD".PRS_CTRL_RST    :=  FALSE;
                   "DV".V1_1_HAND_MODE   :=  FALSE;
                   //switch to next step
                   //-------------------
                   IF (#i > 10) THEN 
                       #step    :=  #step + 50;
                       #i       :=  0;
                   ELSIF "SysTick100ms" THEN
                       #i   :=  #i + 1;
                   END_IF;

               550://start set point ramp of V1 to closed position
                   //---------------------------------------------
                   IF ("KYA".SET_CTL_VALVE_POS > 0.0) THEN
                       IF "SysTick100ms" THEN      
                           "KYA".SET_CTL_VALVE_POS := "KYA".SET_CTL_VALVE_POS - #PRS_CTRL_V1_RMP;
                           IF ("KYA".SET_CTL_VALVE_POS < 0.0) THEN
                               "KYA".SET_CTL_VALVE_POS := 0.0;
                           END_IF;
                       END_IF;
                   ELSE
                       //switch to next step
                       //-------------------
                       IF (#i > 10) THEN 
                           #step    :=  #step + 50;
                           #i       :=  0;
                       ELSIF "SysTick100ms" THEN
                           #i   :=  #i + 1;
                       END_IF;
                   END_IF;        

               600://close valve V2.1
                   //---------------- 
                   "DV".V2_1_CL  :=  TRUE;
                   IF "PDI".LS_V2_1_CL THEN
                       //switch to next step
                       //-------------------
                       IF (#i > 30) THEN 
                           #step    :=  #step + 100;
                           #i       :=  0;
                       ELSIF "SysTick100ms" THEN
                           #i   :=  #i + 1;
                       END_IF;
                   END_IF;       

               700://open V22 for configured blowback duration 
                   //-----------------------------------------
                   IF NOT #fill_up_sto_tank THEN    //fill up already done, set V22 open request
                       "DV".V22_OP   :=  TRUE;
                   END_IF;
                   //blowback
                   //--------
                   IF "PDO".V22  THEN 
                       //count blowbacks
                       //---------------
                       IF ((#i > "CNF".V22_OP_TME) OR ("DIS".ACT_PRS_AR_VSL <= "CNF".MIN_PRS_AR_VSL)) THEN
                           #count   :=  #count + 1;
                           #step    :=  #step + 10;
                           #i       :=  0;
                       ELSE
                           //increase open time
                           //------------------
                           #i   :=  #i + "SY".OB1_PREV_CYCLE;
                       END_IF;
                   END_IF;

               710://close V22
                   //---------
                   "DV".V22_OP   :=  FALSE;
                   //valve closed
                   //------------
                   IF NOT "PDO".V22 THEN
                       //check amount of pulses after two seconds wait time
                       //--------------------------------------------------
                       IF (#i > 20) THEN
                           IF (#count < "CNF".AMT_OF_V22_BB) THEN 
                               #step    :=  #step + 10;
                           ELSE
                               #step    :=  #step + 30;
                           END_IF;
                           #i   :=  0;
                       ELSIF "SysTick100ms" THEN
                           #i := #i + 1;
                       END_IF;
                   END_IF; 

               720://request fill up of gas storage tank
                   //-----------------------------------
                   #fill_up_sto_tank    :=  true;
                   #step                :=  #step + 10;
                   #i                   :=  0;

               730://wait untill fill up of storage tank is done
                   //-------------------------------------------
                   IF NOT #fill_up_sto_tank THEN
                       //wait two seconds after tank filled
                       //----------------------------------
                       IF (#i > 20) THEN
                           #step    :=  #step - 30;
                           #i       :=  0;
                       ELSIF "SysTick100ms" THEN
                           #i := #i + 1;
                       END_IF;
                   END_IF;   

               740://wait 10 seconds
                   //---------------
                   //determine wait time pumping with bypass filter
                   //----------------------------------------------
                   IF (REAL_TO_INT("KYA".WAIT_TME_WITH_BYP_FIL) > 0) THEN
                       #k   :=  REAL_TO_INT("KYA".WAIT_TME_WITH_BYP_FIL / 2 * 60);    // wait time selectable - time base is 2 seconds
                   ELSE
                       #k   :=  5;                                                  // wait time 10s - time base is 2 seconds
                   END_IF;

                   //increase step counter
                   //---------------------
                   IF (#i > #k) THEN   
                       #step    :=  #step + 60;
                       #i       :=  0;
                   //count wait time
                   //----------------
                   ELSIF "SysTick2s" THEN
                       #i   :=  #i + 1;
                   END_IF;

               800://pump down main filter after flushing
                   //------------------------------------                   
                   "DV".V3_3_OP := TRUE;       //open valve V3.3

                   IF "PDI".LS_V3_3_OP THEN
                       #step    :=  #step + 100;
                   END_IF;            

               900://check if main filter pressure reached furnace pressure
                   //------------------------------------------------------
                   IF ("DIS".ACT_PRS_CLF >= "DIS".ACT_PRS_MAIN_FIL) THEN  
                       "DV".V3_3_OP  := FALSE;     //close valve V3.3
                       IF "PDI".LS_V3_3_CL THEN 
                           IF "SysTick100ms" THEN
                               #i   :=  #i + 1;
                           END_IF;
                           //open valve V2.1
                           //---------------
                           IF (#i > 10) THEN   
                               "DV".V2_1_CL := FALSE;
                               #step    :=  #step + 100;
                               #i       :=  0;
                           END_IF;
                       END_IF;
                     END_IF;

              1000://hold set point of valve V1.1 
                   //----------------------------
                   IF "PDI".LS_V2_1_OP THEN 
                       "DV".V1_1_HAND_MODE:= TRUE;
                       //switch to next step
                       //-------------------
                       IF (#i > 10) THEN 
                           #step    :=  #step + 100;
                           #i       :=  0;
                       ELSIF "SysTick100ms" THEN
                           #i   :=  #i + 1;
                       END_IF;
                   END_IF; 

              1100://reset pressure controller output
                   //--------------------------------
                   //switch to next step
                   //-------------------
                   IF (#i > 10) THEN 
                       #step    :=  #step + 100;
                       #i       :=  0;
                   ELSIF "SysTick100ms" THEN
                       "KYD".PRS_CTRL_RST    :=  TRUE;
                       #i   :=  #i + 1;
                   END_IF;

              1200://transfer pressure control output to set point of V1
                   //---------------------------------------------------
                   "KYD".PRS_CTRL_RST    :=  FALSE;
                   "DV".V1_HAND_MODE     :=  FALSE;
                   //switch to next step
                   //-------------------
                   IF (#i > 10) THEN 
                       #step    :=  #step + 100;
                       #i       :=  0;
                   ELSIF "SysTick100ms" THEN
                       #i   :=  #i + 1;
                   END_IF;

              1300://start set point ramp of V1.1 to closed position
                   //-----------------------------------------------
                   IF ("KYA".SET_CTL_VALVE_POS_V1_1 > 0.0) THEN
                       IF "SysTick100ms" THEN      
                           "KYA".SET_CTL_VALVE_POS_V1_1 := "KYA".SET_CTL_VALVE_POS_V1_1 - #PRS_CTRL_V1_1_RMP;
                           IF ("KYA".SET_CTL_VALVE_POS_V1_1 < 0.0) THEN
                               "KYA".SET_CTL_VALVE_POS_V1_1 := 0.0;
                           END_IF;
                       END_IF;
                   ELSE
                       //switch to next step
                       //-------------------
                       IF (#i > 10) THEN
                           IF (("STA".ACT_DVC_CNF_BYTE_3 AND 2#0010_0000) = 2#0010_0000) THEN 
                               #step    :=  #step + 200;     //without bypass filter
                           ELSE     
                               #step    :=  #step + 100;     //with bypass filter
                               #i       :=  0;
                           END_IF;

                       ELSIF "SysTick100ms" THEN
                           #i   :=  #i + 1;
                       END_IF;
                   END_IF;        

              1400://close valve V2.11
                   //----------------- 
                   "DV".V2_11_OP :=  FALSE;
                   IF "PDI".LS_V2_11_CL THEN
                       //switch to next step
                       //-------------------
                       IF (#i > 30) THEN 
                           #step    :=  #step + 100;
                           #i       :=  0;
                       ELSIF "SysTick100ms" THEN
                           #i   :=  #i + 1;
                       END_IF;
                   END_IF;       

              1500://vent bypass filter with Ar or watercooled bypass tube installed
                   //---------------------------------------------------------------
                   IF ("DV".APS_BY_FIL_DELAYED OR (("STA".ACT_DVC_CNF_BYTE_3 AND 2#0010_0000) = 2#0010_0000)) THEN 
                       "DV".V22_1_OP         := FALSE;
                       "DV".P3_ON            := FALSE;       //switch pump P3 off
                       #fil_cln_req_in_prc  := FALSE;
                       "LT".ABORT_FIL_CLN    := FALSE;
                       "LT".SI_FIL_FSH_SEQ_ON:= FALSE;
                       "FLT".SI_FIL_REG_ENB  := FALSE;
                   ELSE
                       "DV".V22_1_OP := TRUE;
                   END_IF;   

              2000://sequence aborted - initialisation
                   //---------------------------------
                   #i                   := 0;
                   #fill_up_sto_tank    := false;       //reset flag fill up sequence storage tank 
                   "DV".V22_OP           := FALSE;
                   "DV".V22_1_OP         := FALSE;
                   "DV".V25_OP           := FALSE;
                   "DV".V3_4_OP          := FALSE;
                   "DV".V1_HAND_MODE     := TRUE;        //V1 keeps last KYA set point
                   #step                := #step + 100;

              2100://sequeunce aborted - switch back to main pump line
                   //-------------------------------------------------
                   //valve V2.1 is closed
                   //--------------------
                   IF "DV".V2_1_CL THEN
                       //furnace pressure is above main filter pressure
                       //----------------------------------------------
                       IF ("DIS".ACT_PRS_CLF > "DIS".ACT_PRS_MAIN_FIL) THEN 
                           IF (#i > 10) THEN        //1 sec delay for closing V3.3
                               "DV".V3_3_OP  := FALSE;
                           ELSIF "SysTick100ms" THEN
                               #i   :=  #i + 1;
                           END_IF;

                           //pump down valve main filter to P3 is closed
                           //-------------------------------------------
                           IF "PDI".LS_V3_3_CL THEN   
                               "DV".V2_1_CL              :=  FALSE;  //open valve V2.1 to main filter
                               "KYA".SET_CTL_VALVE_POS   :=  50.0;   //set initial set point of V1
                               #i                       :=  0;
                           END_IF;

                       //furnace pressure is below main filter pressure
                       //----------------------------------------------
                       ELSE 
                           "DV".V3_3_OP  := TRUE;        //pump down main filter
                       END_IF;
                   //valve V2.1 is opened
                   //--------------------
                   ELSE
                       //close bypass line
                       //-----------------
                       "DV".V2_11_OP                 :=  FALSE;      //close V2.11
                       "DV".V1_1_HAND_MODE           :=  TRUE;       //close V1.1
                       "KYA".SET_CTL_VALVE_POS_V1_1  :=  0.0;

                       //switch to next step
                       //-------------------
                       IF (#i > 30) THEN            //3 sec delay for switching to next step
                           #step    := #step + 100;
                           #i       := 0;
                       ELSIF "SysTick100ms" THEN
                           #i   :=  #i + 1;
                       END_IF;

                   END_IF;

              2200://sequeunce aborted - switch back to main pump line
                   //-------------------------------------------------
                   IF (#i > 10) THEN 
                       "DV".V1_HAND_MODE     := FALSE;       //set pressure control out to set point of V1
                       "KYD".PRS_CTRL_RST    := FALSE;       
                       #step                := 1500;        //switch to step 1500 and finish sequence
                   ELSIF "SysTick100ms" THEN
                       "KYD".PRS_CTRL_RST    := TRUE;        //reinitialize pressure controller
                       #i   :=  #i + 1;
                   END_IF;
           END_CASE;

       ELSE

           #step    :=  0;      //reset step counter
           //keep valves of bypass line closed
           //---------------------------------
           "DV".V2_11_OP                 :=  FALSE;
           "DV".V1_1_HAND_MODE           :=  TRUE;
           "KYA".SET_CTL_VALVE_POS_V1_1  :=  0.0;
           "DV".V3_3_OP                  :=  FALSE;
           "DV".V3_4_OP                  :=  FALSE;
           "LT".ABORT_FIL_CLN            :=  FALSE;
           "DV".V22_OP                   :=  FALSE;
           "DV".V22_1_OP                 :=  FALSE;
           "DV".P3_ON                    :=  FALSE;
           //disable hand mode of valve V1
           //-----------------------------
           "DV".V1_HAND_MODE             :=  FALSE;

       END_IF;

       //delay reset of filter cleaning request
       //--------------------------------------
       "DV".FIL_CLN_REQ_IN_PRC   := "SysOffdelay"( DIN     := #fil_cln_req_in_prc,
                                               SetTime := 5,                           // setp. time
                                               ActTime := #fil_cln_off_dly,             // act. time
                                               Tick    := "SysTick100ms");               // timebase (100ms)
END_FUNCTION_BLOCK

FUNCTION_BLOCK "PM_DRV_COMM_LZI950"   // FB507, SCL
{ S7_Optimized_Access := 'FALSE' }
VERSION : 0.0
// --------------------------------------------------------------------------------
//     program     :    PM_DRV_COMM_LZI950
//     description :    communication with Lenze i950 
//     
//     name        :    L. Ewert
//     date        :    28.08.2018
// 
//     revision    :
//     name        :
//     date        :    
//                     (c)PVATepla
//     --------------------------------------------------------------------------------
   VAR_INPUT
      Enable : Bool;   // Enable or disable the controller (will set the brake if used)
      Pro_start : Bool;   // For any speed or position control you have to use a profile and edit the speed
      Speed_ext_ovr : Bool;   // Has to be TRUE if you want to change the speed of the profile
      Ref_Start : Bool;   // Trigger a ref. process (Positive edge)
      Ref_reset : Bool;   // Reset the ref. of the drive now you can start a new ref
      Reset_error : Bool;   // Reset any error of the Drive
      Stop : Bool;   // End a Profile movement (stops the drive)
      Profil : Int;   // Profil from 1-15 0 = No movement possible
      PM_ADR_E : Word;   // Adress has to be in Hex form.
      PM_ADR_A : Word;   // Adress has to be in Hex form.
      Units_per_rev : Real;   // A value in the controller for 1 turn of the drive
      Gear_ratio : Real;   // Gear ratio for the calculation of the set speed in Units/sec Bsp: drive = 10 re
      Set_vel : Real;   // Speed in Rounds per min. after gear (so the drive speed will be calculated with
   END_VAR
   VAR_OUTPUT
      Standstill : Bool;   // Drive vel = 0
      Error : Bool;   // An Error form the drive controller is been set
      Ref_Done : Bool;   // Ref. is been done so the drive does have a valid position
      Busy : Bool;   // Drive is doing an action (Ref or Profile is activ)
      LS_neg : Bool;   // DI of LS neg is been set
      LS_pos : Bool;   // DI of LS pos is been set
      Ready : Bool;   // Ready drive is ready for movement
      Pos_cont_active : Bool;   // Movement in pos. direction
      Error_code : DInt;   // Error code from Lenze
      Act_pos : Real;   // Actual position of the drive
      Act_vel : Real;   // Actual velocity of the drive after gear (so should be the same as the set_vel)
   END_VAR
   VAR
      DRV_DATA_LZ_I950 : "UDT_DRV_LENZE_i950";
      Switch_on : Bool := TRUE;
      Ref_vel_override : Bool := TRUE;
      counter_FB : Int;
      counter_1 : Int;
      Error_Write_Data : Int;
      Error_Read_Data : Int;
      Switch_on_time : Int;
      Enable_on_time : Int;
      Vel_in_Units_sec : Real;
   END_VAR
   VAR_TEMP
      Profil_tmp : Byte;
   END_VAR
BEGIN

       // Because the drive is probably having an error it is been reset after starting it  
       IF "SysTick100ms" AND #Switch_on THEN
           #counter_1 := #counter_1+1;
           IF #counter_1 >= 30 THEN
               #Switch_on:= FALSE;
           END_IF;
       END_IF;
       IF #Gear_ratio = 0 THEN 
           #Gear_ratio := 1; 
       END_IF;
       IF #Units_per_rev = 0 THEN
           #Units_per_rev := 1.0;
       END_IF;

       // Read Drive Data into Struct
       #Error_Read_Data := DPRD_DAT ( LADDR := #PM_ADR_E, 
                                     RECORD=> #DRV_DATA_LZ_I950.Input);                              

       // Write Input Data to Drive Data
       #DRV_DATA_LZ_I950.Output.Control_Bools.Enable := #Enable;
       IF NOT #Enable THEN
           #Enable_on_time:= 0;
       END_IF;
       // Because the drive is only valuating signals after it is enabled 
       // it is important to wait till it is running before sending any controls
       IF #Enable AND #Enable_on_time < 10 THEN
           IF "SysTick100ms" THEN
               #Enable_on_time:= #Enable_on_time+1;
           END_IF;
       ELSE 
           #DRV_DATA_LZ_I950.Output.Control_Bools.Do_pos_drv    := #Pro_start AND NOT #Stop;
           #DRV_DATA_LZ_I950.Output.Control_Bools.Enab_ext_vel  := #Speed_ext_ovr;
           #DRV_DATA_LZ_I950.Output.Control_Bools.Start_homing  := #Ref_Start;    
           #DRV_DATA_LZ_I950.Output.Control_Bools.Reset_ref_pos := #Ref_reset;
           #DRV_DATA_LZ_I950.Output.Control_Bools.Res_error     :=(#Reset_error OR #Switch_on) AND #DRV_DATA_LZ_I950.Input.Status_Bools_1.Standstill OR #DRV_DATA_LZ_I950.Input.Status_Bools_1.Drv_error;
           #DRV_DATA_LZ_I950.Output.Control_Bools.Stop          := #Stop;
           // Convert Profil Nr. to 4 Bit coded Profil Nr. Bsp: 0010 = 2 // 1010 = 10 usw.
           IF #Profil > 15 THEN #Profil := 15; END_IF;
           #Profil_tmp := INT_TO_BYTE(#Profil);
           #DRV_DATA_LZ_I950.Output.Control_Bools.Profile_BIT_0 := BYTE_TO_BOOL(#Profil_tmp AND 2#0000_0001);
           #DRV_DATA_LZ_I950.Output.Control_Bools.Profile_BIT_1 := BYTE_TO_BOOL(SHR(IN:=#Profil_tmp,N:=1) AND 2#0000_0001);
           #DRV_DATA_LZ_I950.Output.Control_Bools.Profile_BIT_2 := BYTE_TO_BOOL(SHR(IN:=#Profil_tmp,N:=2) AND 2#0000_0001);
           #DRV_DATA_LZ_I950.Output.Control_Bools.Profile_BIT_3 := BYTE_TO_BOOL(SHR(IN:=#Profil_tmp,N:=3) AND 2#0000_0001);
       END_IF;
       IF #Gear_ratio <> 0 THEN 
           // Calculate Vel from Rpm to Units/sec -> 1 round -> 36.0000 Digits /// RPS Drive = (RPM(after gear) * 10000 (Digits after point 0.0000) / (60 (Min into Sec) * Gear_Ratio)) * Units per Revolution 
           #Vel_in_Units_sec := ((#Set_vel * 10000.0) / (60.0 * #Gear_ratio)) * #Units_per_rev;
       END_IF;
       #DRV_DATA_LZ_I950.Output.Control_Para.Ext_vel := DINT_TO_DWORD(REAL_TO_DINT(#Vel_in_Units_sec));

       // Write Struct to Drive Data
       #Error_Write_Data := DPWR_DAT ( LADDR := #PM_ADR_A, 
                                      RECORD:= #DRV_DATA_LZ_I950.Output);

       // Set Outputs                              
       #Standstill  := #DRV_DATA_LZ_I950.Input.Status_Bools_1.Standstill;
       #Error       := #DRV_DATA_LZ_I950.Input.Status_Bools_1.Drv_error OR #DRV_DATA_LZ_I950.Input.Status_Bools_1.STO_active;                               
       #Ref_Done    := #DRV_DATA_LZ_I950.Input.Status_Bools_1.Homing_finished;
       #Busy        := #DRV_DATA_LZ_I950.Input.Status_Bools_1.Homing_active OR #DRV_DATA_LZ_I950.Input.Status_Bools_1.Jog_active
                       OR #DRV_DATA_LZ_I950.Input.Status_Bools_1.Pos_cont_active;
       #LS_neg      := #DRV_DATA_LZ_I950.Input.Status_Bools_1.LS_neg;
       #LS_pos      := #DRV_DATA_LZ_I950.Input.Status_Bools_1.LS_pos;
       #Ready       := #DRV_DATA_LZ_I950.Input.Status_Bools_1.Drv_ready AND #DRV_DATA_LZ_I950.Input.Status_Bools_1.Op_enabled;
       #Pos_cont_active := #DRV_DATA_LZ_I950.Input.Status_Bools_1.Pos_cont_active;
       #Error_code  := DWORD_TO_DINT(DW#16#0000FFFF AND #DRV_DATA_LZ_I950.Input.Status_Para.Error_code); // The high Word is used from LENZE only so we don't need it 
                                                                                                       // All Errors can be detected by using the lower Byte

       // Shift 4 digits of the DWORD Value so they appear after the decimal point Pos is the actual Drive pos not the pos after gear !!!!
       #Act_pos     := (DINT_TO_REAL(DWORD_TO_DINT(#DRV_DATA_LZ_I950.Input.Status_Para.Act_pos))* #Gear_ratio / (#Units_per_rev *10000.0));

       IF #Units_per_rev <> 0 THEN
           // Calculate Vel from Units/sec -> RPM after Gear -->> 36.0000 Units/per rev. // RPM After Gear = RPS(from drive) * 60 (Sec into Min) * Gear_Ratio / ((Units_per_revolution) * 10000) (Digits after point 0.0000)
           #Act_vel := DINT_TO_REAL(DWORD_TO_DINT(#DRV_DATA_LZ_I950.Input.Status_Para.Act_vel)) * #Gear_ratio * 60.0 / (#Units_per_rev * 10000.0);
       END_IF;
END_FUNCTION_BLOCK

FUNCTION "FLT_BLKMOV" : Void   // FC3, STL
TITLE = Coppy all fault bits into data of CDP
{ S7_Optimized_Access := 'FALSE' }
VERSION : 0.1
   VAR_TEMP
      RETVAL : Int;
   END_VAR
BEGIN

REGION Network 1
         CALL  BLKMOV
         ( SRCBLK  := P#DB142.DBX0.0 BYTE 68,
           RET_VAL := #RETVAL,
           DSTBLK  := P#DB636.DBX0.0 BYTE 68
         );
END_REGION
END_FUNCTION

FUNCTION "CM_ITL_IO" : Void   // FC67, SCL
{ S7_Optimized_Access := 'FALSE' }
VERSION : 0.0
// --------------------------------------------------------------------------------
//     program     :    CM_ITL_IO
//     description :    Interlock modul        
//     name        :    L. Vogel
//     date        :    19.12.12
// 
//     revision    :
//     name        :    
//     date        :   
//                     (c)CGS
//     --------------------------------------------------------------------------------
   VAR_INPUT
      ADR : Int;
      KYD_ON : Bool;
      KYD_OFF : Bool;
      AUTO : Bool;
      DC_ON : Bool;
      CON1 : Bool;
      CON2 : Bool;
      CON3 : Bool;
      CON4 : Bool;
      CON5 : Bool;
      CON6 : Bool;
      CON7 : Bool;
      CON8 : Bool;
   END_VAR
   VAR_IN_OUT
      LT_OUT : Bool;
      ITL_OUT : Word;
   END_VAR
   VAR_TEMP
      ITL : Byte;
      ITL_BIT AT ITL : Array[0..7] of Bool;
   END_VAR
BEGIN

   #ITL_BIT[0] := #CON1;
   #ITL_BIT[1] := #CON2;
   #ITL_BIT[2] := #CON3;
   #ITL_BIT[3] := #CON4;
   #ITL_BIT[4] := #CON5;
   #ITL_BIT[5] := #CON6;
   #ITL_BIT[6] := #CON7;
   #ITL_BIT[7] := #CON8;

   IF #ITL = 2#11111111 THEN
       IF #AUTO THEN
           #LT_OUT := #DC_ON;
       ELSE
           #LT_OUT := (#LT_OUT OR #KYD_ON) AND NOT #KYD_OFF;
       END_IF;
   ELSE
       #LT_OUT := FALSE;
       IF #KYD_ON AND NOT #AUTO THEN
           #ITL_OUT := BYTE_TO_WORD(#ITL) OR SHL(IN:=INT_TO_WORD(#ADR),N:=8);
       END_IF;
   END_IF;
END_FUNCTION

FUNCTION "PM_CALL_ST" : Void   // FC90, SCL
{ S7_Optimized_Access := 'FALSE' }
VERSION : 0.0
BEGIN

       "PM_HAI"();                          //Read analog inputs
       "PM_DI_DB"();                  //call digital input module
       "PM_DO_DB"();                  //call digital output module
       "PM_AI_DB"();                  //call analog input module
       "PM_AO_DB"();                  //call analog output module
       "PM_HAO"();                          //Write analog Outputs

       "PM_MDI_DB"();          //call digital input module service mode
       "PM_MDO_DB"();          //call digital output module service mode
       "PM_MAI_DB"();          //call analog input module service mode
       "PM_MAO_DB"();          //call analog output module service mode

       "PM_GET_POS"();                      //get all positions   
       "PM_GET_WGT_XT_CLP_DB"();
       "DIS".ACT_PLT_HDW_ID  := 1.0;
END_FUNCTION

FUNCTION "PM_AI_CONVERT" : Real   // FC92, SCL
{ S7_Optimized_Access := 'FALSE' }
VERSION : 0.0
// --------------------------------------------------------------------------------
//     program     :    PM_AI_CONVERT
//     description :    fetch, convert and scale  analog input signal       
//     name        :    K. Kalkowski
//     date        :    08.12.98
// 
//     revision    :    add convert type 3
//     name        :    G. Eibelsh鋟ser
//     date        :    14.12.99
//     
//     revision    :    add convert type 6
//     name        :    G. Eibelsh鋟ser
//     date        :    05.06.00
//     
//     revision    :    add convert type 7 and 8
//     name        :    G. Eibelsh鋟ser
//     date        :    28.09.00
//     
// 
//                     (c)CGS
//     --------------------------------------------------------------------------------
   VAR_INPUT
      CHANNEL : Real;
      CONVERT_PAR : Struct
         hardware_type : Int;
         convert_type : Int;
         min_value : Real;
         max_value : Real;
      END_STRUCT;
   END_VAR
   VAR_TEMP
      input_real : Real;
      max_range : Real;
      min_range : Real;
      max_range_current : Real;
      min_range_current : Real;
      max_range_voltage : Real;
      min_range_voltage : Real;
   END_VAR
BEGIN


       #input_real := #CHANNEL;               //fetch input

       IF #CONVERT_PAR.convert_type = 0 THEN                   // spare input 

           #input_real := 0.0;   

           #PM_AI_CONVERT := #input_real;                       //set return value

       END_IF;

       IF #CONVERT_PAR.convert_type = 1 THEN                   // ai_type 1 [-1.0..1.0/lin] 

           #max_range := 1.0;                                  //input limits 
           #min_range := -1.0;
           IF #input_real > #max_range THEN
               #input_real := #max_range; 
           END_IF;
           IF #input_real < #min_range THEN
               #input_real := #min_range; 
           END_IF;
           //calculate input value 
           #input_real := (#input_real-#min_range)/(#max_range-#min_range)*(#CONVERT_PAR.max_value-#CONVERT_PAR.min_value)+#CONVERT_PAR.min_value;   

           #PM_AI_CONVERT := #input_real;                       //set return value

       END_IF;

       IF #CONVERT_PAR.convert_type = 2 THEN                   // ai_type 2 [0.0..1.0/lin] 

           #max_range := 1.0;                                  //input limits 
           #min_range := 0.0;
           IF #input_real > #max_range THEN
               #input_real := #max_range; 
           END_IF;
           IF #input_real < #min_range THEN
               #input_real := #min_range; 
           END_IF;
           //calculate input value 
           #input_real := (#input_real-#min_range)/(#max_range-#min_range)*(#CONVERT_PAR.max_value-#CONVERT_PAR.min_value)+#CONVERT_PAR.min_value;   

           #PM_AI_CONVERT := #input_real;                       //set return value

       END_IF;

       IF #CONVERT_PAR.convert_type = 3 THEN                   // ai_type 3 [0.0..1.0]

           #max_range := 1.0;                                  //input limits 
           #min_range := 0.0;

           #max_range_current    :=150;                        //max. output sensor signal 150yA
           #min_range_current    :=0;

           IF #input_real > #max_range THEN
               #input_real := #max_range; 
           END_IF;
           IF #input_real < #min_range THEN
               #input_real := #min_range; 
           END_IF;


           //calculate input value 
           #input_real := (#input_real-#min_range)/(#max_range-#min_range)*(#max_range_current-#min_range_current)+#min_range_current; 

           //Call Linearisation function and set return value

           #PM_AI_CONVERT    :="PM_LINEARISATION"         
                             (x        := #input_real,
                              x_data   := "PM_DEVICE_IRCON_R727".signal,   // array with x values
                              y_data   := "PM_DEVICE_IRCON_R727".temp);    // array with y values

       END_IF;

       IF #CONVERT_PAR.convert_type = 4 THEN                   // ai_type 4 [0.0..1.0]

           #max_range := 1.0;                                  //input limits 
           #min_range := 0.0;

           #max_range_voltage    :=50;                         //max. output sensor signal 50mV
           #min_range_voltage    :=0;

           #input_real := (#input_real * 1.2);

           IF #input_real > #max_range THEN
               #input_real := #max_range; 
           END_IF;
           IF #input_real < #min_range THEN
               #input_real := #min_range; 
           END_IF;


           //calculate input value 
           #input_real := (#input_real-#min_range)/(#max_range-#min_range)*(#max_range_voltage-#min_range_voltage)+#min_range_voltage; 

           //Call Linearisation function and set return value

           #PM_AI_CONVERT    :="PM_LINEARISATION"         
                             (x        := #input_real,
                              x_data   := "PM_DEVICE_IRCON_11x20".signal,   // array with x values
                              y_data   := "PM_DEVICE_IRCON_11x20".temp);    // array with y values


       END_IF;

       IF #CONVERT_PAR.convert_type = 5 THEN                   // ai_type 5 [0.0..1.0] 

           #max_range := 1.0;                                  //input limits 
           #min_range := 0.0;
           IF (#input_real * 10.0 / 7.0) > #max_range THEN
               #input_real := #max_range; 
           END_IF;
           IF (#input_real * 10.0 / 7.0) < #min_range THEN
               #input_real := #min_range; 
           END_IF;

           //calculate input value
           //lifted to 143% of full scale                     
           #input_real := (10.0 / 7.0 * #input_real-#min_range)/(#max_range-#min_range)*(#CONVERT_PAR.max_value-#CONVERT_PAR.min_value)+#CONVERT_PAR.min_value;   

           #PM_AI_CONVERT := #input_real;                       //set return value

       END_IF;

       IF #CONVERT_PAR.convert_type = 6 THEN                   // ai_type 6 [0.0..1.0] 

           #max_range := 1.0;                                  //input limits 
           #min_range := 0.0;
           IF (#input_real * 2.0) > #max_range THEN
               #input_real := #max_range; 
           END_IF;
           IF (#input_real * 2.0) < #min_range THEN
               #input_real := #min_range; 
           END_IF;

           //calculate input value
           //lifted to 200 % of full scale                    
           #input_real := (2.0 * #input_real-#min_range)/(#max_range-#min_range)*(#CONVERT_PAR.max_value-#CONVERT_PAR.min_value)+#CONVERT_PAR.min_value;   

           #PM_AI_CONVERT := #input_real;                       //set return value

       END_IF;

       IF #CONVERT_PAR.convert_type = 7 THEN                   // ai_type 7 [0.19..1.0] 

           #max_range := 1.0;                                  //input limits 
           #min_range := 0.19;                                 
           IF #input_real > #max_range THEN
               #input_real := #max_range; 
           END_IF;
           IF #input_real < #min_range THEN
               #input_real := #min_range; 
           END_IF;

           //calculate input value
           //find formula in Thermovac manual 
           #input_real := (10**((10 * #input_real - 6.143) / 1.286));   

           #PM_AI_CONVERT := #input_real;                       //set return value

       END_IF;

       IF #CONVERT_PAR.convert_type = 8 THEN                   // ai_type 8 [0.2..1.0/lin] 

           #max_range := 1.0;                                  //input limits 
           #min_range := 0.2;                                  // !! min limit 0.2 
           IF #input_real > #max_range THEN
               #input_real := #max_range; 
           END_IF;
           IF #input_real < #min_range THEN
               #input_real := #min_range; 
           END_IF;
           //calculate input value 
           #input_real := (#input_real-#min_range)/(#max_range-#min_range)*(#CONVERT_PAR.max_value-#CONVERT_PAR.min_value)+#CONVERT_PAR.min_value;   

           #PM_AI_CONVERT := #input_real;                       //set return value

       END_IF;

       IF #CONVERT_PAR.convert_type = 9 THEN                   // ai_type 7 [0.19..1.0] 

           #max_range := 0.868;                                  //input limits 
           #min_range := 0.22;                                 
           IF #input_real > #max_range THEN
               #input_real := #max_range; 
           END_IF;
           IF #input_real < #min_range THEN
               #input_real := #min_range; 
           END_IF;

           //calculate input value
           //find formula in pfeiffer PCR280 manual 
           #input_real := (10**(10 * #input_real - 5.5));   

           #PM_AI_CONVERT := #input_real;                       //set return value

       END_IF;
END_FUNCTION

FUNCTION "PM_AO_CONVERT" : Real   // FC93, SCL
{ S7_Optimized_Access := 'FALSE' }
VERSION : 0.0
// --------------------------------------------------------------------------------
//     program     :    PM_AO_CONVERT
//     description :    convert, scale and write analog output signal       
//     name        :    K. Kalkowski
//     date        :    17.12.98
//     
//     revision    :
//     name        :
//     date        :    
//                     (c)CGS
//     --------------------------------------------------------------------------------
   VAR_INPUT
      OUTVALUE : Real;
      CONVERT_PAR : Struct
         hardware_type : Int;
         convert_type : Int;
         min_value : Real;
         max_value : Real;
      END_STRUCT;
   END_VAR
   VAR_TEMP
      output_real : Real;
      max_range : Real;
      min_range : Real;
   END_VAR
BEGIN


       #output_real := #OUTVALUE;                               //fetch output value

       IF #output_real > #CONVERT_PAR.max_value THEN            //input limits
               #output_real := #CONVERT_PAR.max_value; 
           END_IF;
           IF #output_real < #CONVERT_PAR.min_value THEN
               #output_real := #CONVERT_PAR.min_value; 
           END_IF;

       IF #CONVERT_PAR.convert_type = 0 THEN                   // spare output

           #output_real := 0.0;

       END_IF;       

       IF #CONVERT_PAR.convert_type = 1 THEN                   // ao_type 1 [-1.0..1.0/lin] 

           #max_range := 1.0;                                  //set output range                                  
           #min_range := -1.0;
                                                              //calculate output value 
           #output_real := (#output_real-#CONVERT_PAR.min_value)/(#CONVERT_PAR.max_value-#CONVERT_PAR.min_value)*(#max_range-#min_range)+#min_range;   

       END_IF;

       IF #CONVERT_PAR.convert_type = 2 THEN                   // ao_type 2 [0.0..1.0/lin] 

           #max_range := 1.0;                                  //set output range 
           #min_range := 0.0;
                                                              //calculate output value
           #output_real := (#output_real-#CONVERT_PAR.min_value)/(#CONVERT_PAR.max_value-#CONVERT_PAR.min_value)*(#max_range-#min_range)+#min_range;   

       END_IF;

       IF #CONVERT_PAR.convert_type = 3 THEN                   // ao_type 3 [0.0..1.0] 

           #max_range := 1.0;                                  //set output range 
           #min_range := 0.0;

           // 50% of max output                                                             //calculate output value
           #output_real := 0.5 * (#output_real-#CONVERT_PAR.min_value)/(#CONVERT_PAR.max_value-#CONVERT_PAR.min_value)*(#max_range-#min_range)+#min_range;   

       END_IF;


       #PM_AO_CONVERT := #output_real;                          //set return value                                           //set return value
END_FUNCTION

FUNCTION "PM_LINEARISATION" : Real   // FC94, SCL
{ S7_Optimized_Access := 'FALSE' }
VERSION : 0.0
// --------------------------------------------------------------------------------
//     program     :    PM_LINEARISATION
//     description :    fetch real input and linerise between two values 
//     name        :    G. Eibelsh鋟ser
//     date        :    09.12.99 
//     
//     revision    :  
//     name        :  
//     date        :  
//                     (c) CGS
//     --------------------------------------------------------------------------------
   VAR_INPUT
      x : Real;   // signal input
      x_data : Array[1..46] of Real;
      y_data : Array[1..46] of Real;
   END_VAR
   VAR_TEMP
      x1 : Real;
      x2 : Real;
      y1 : Real;
      y2 : Real;
      y : Real;
      i : Int;
      found : Int;
   END_VAR
BEGIN

         #i := 1;                                // search for interval in data list
          #found := 0;

         WHILE #found = 0 DO

           #x1 := #x_data[#i];
           #x2 := #x_data[#i+1];
           #y1 := #y_data[#i];
           #y2 := #y_data[#i+1];

           IF (#x <= #x1) THEN                             // below x1 ?

             #y := #y1;  
             #found := 1;
           ELSE
             IF (#x < #x2) THEN                            // x1<x<x2 ?
                 #y := #y1 + ((#y2-#y1)/(#x2-#x1))*(#x-#x1);
                 #found := 1;
             ELSE

                 IF (#i = 46) THEN                        // last x[i] because i = 46 ?
                   #y := #y2;
                   #found := 1;

                 ELSE
                   #i := #i + 1;                           // next x[i]
                   #found := 0;

                 END_IF;
              END_IF;
             END_IF;
           END_WHILE;

   #PM_LINEARISATION    := #y;
END_FUNCTION

FUNCTION "PM_GET_POS" : Void   // FC96, SCL
{ S7_Optimized_Access := 'FALSE' }
VERSION : 0.0
// --------------------------------------------------------------------------------
//     program:         PM_GET_POS
//     description :    Get all positions and convert to mm or ?
//     name:               lv
//     date        :       20.09.2018
//     
//     revision:        
//     name:           
//     Date:          
// 
//                 (c)PVATepla AG
// --------------------------------------------------------------------------------
   VAR_TEMP
      SET_REF_POS : DWord;
      LS_ENC_PRESET : Bool;
   END_VAR
   VAR CONSTANT
      enc_inc_rot : Int := 4096;
   END_VAR
BEGIN

       // Crystal handling swivel in [癩
       "AV".XT_HDL_SW_ENC_POS := (DINT_TO_REAL(DWORD_TO_DINT("P_BM_XT_HDL_SW_ENC_POS":P))/#enc_inc_rot* "CNF".XT_HDL_SW_ENC_RATIO)-90.0; // 90,0=Offset encoder value 
       #SET_REF_POS := DINT_TO_DWORD(REAL_TO_DINT(("CNF".XT_HDL_SW_REF_POS+90.0)/"CNF".XT_HDL_SW_ENC_RATIO* #enc_inc_rot));
       IF "DV".XT_HDL_SW_SET_REF_POS  THEN
           "TI_PRESET_XT_HDL_SW"  := "TI_PRESET_XT_HDL_SW" + 1;
           "P_BM_XT_HDL_SW_ENC_REF":P := #SET_REF_POS OR 2#1000_0000_0000_0000_0000_0000_0000_0000;
       ELSE
           "TI_PRESET_XT_HDL_SW"  := 0;
           "P_BM_XT_HDL_SW_ENC_REF":P := 16#0000_0000;
       END_IF;

       "DV".XT_HDL_SW_SET_REF_POS := "KYD".XT_HDL_SW_REF_RES OR (("VIMP_LS_XT_HDL_SW_LOCK">0) AND ("VIMP_LS_XT_HDL_SW_LOCK"<4)) ;

       IF "PDI".LS_XT_HDL_SW_LOCK THEN
           IF "SysTick1s" AND "VIMP_LS_XT_HDL_SW_LOCK"<4 THEN
              "VIMP_LS_XT_HDL_SW_LOCK" := "VIMP_LS_XT_HDL_SW_LOCK" +1;
           END_IF;    
       ELSE    
           "VIMP_LS_XT_HDL_SW_LOCK" := 0;
       END_IF;    

       // Furnace chamber lift in [mm]
       "AV".FCH_ENC_POS := (DINT_TO_REAL(DWORD_TO_DINT("P_BM_FCH_ENC_POS":P))/#enc_inc_rot * "CNF".FCH_ENC_RATIO-120.0); // 100,0=Offset encoder value
       #SET_REF_POS    := DINT_TO_DWORD(REAL_TO_DINT(("CNF".FCH_REF_POS+100.0)/"CNF".FCH_ENC_RATIO* #enc_inc_rot));    
       IF "DV".FCH_SET_REF_POS THEN
           "TI_PRESET_FCH_LFT"  := "TI_PRESET_FCH_LFT" - 1;
          "P_BM_FCH_ENC_REF":P := #SET_REF_POS OR 2#1000_0000_0000_0000_0000_0000_0000_0000;    
       ELSE 
          "P_BM_FCH_ENC_REF":P := 16#0000_0000;;
       END_IF;

       "DV".FCH_SET_REF_POS := "KYD".FCH_LFT_REF_SET;

       // technolgy flange lift in [mm]
       "AV".TEC_FLG_ENC_POS := (DINT_TO_REAL(DWORD_TO_DINT("P_BM_TEC_FLG_ENC_POS":P))/#enc_inc_rot * "CNF".TEC_FLG_ENC_RATIO)-120.0; // 100,0=Offset encoder value
       #SET_REF_POS := DINT_TO_DWORD(REAL_TO_DINT(("CNF".TEC_FLG_REF_POS+100.0)/"CNF".TEC_FLG_ENC_RATIO* #enc_inc_rot));
       IF "DV".TEC_FLG_SET_REF_POS THEN
          "TI_PRESET_TEC_FLG"  := "TI_PRESET_TEC_FLG"-1;
          "P_BM_TEC_FLG_ENC_REF":P    := #SET_REF_POS OR 2#1000_0000_0000_0000_0000_0000_0000_0000;
       ELSE 
          "P_BM_TEC_FLG_ENC_REF":P    := 16#0000_0000;
       END_IF;

       "DV".TEC_FLG_SET_REF_POS := (("TI_PRESET_TEC_FLG">0) AND ("TI_PRESET_TEC_FLG"<4)) OR "KYD".TEC_FLG_LFT_REF_SET;  

       IF "PDI".LS_TEC_FLG_DN AND NOT "PFM_TEC_FLG_DN" THEN  
          "PFM_TEC_FLG_DN" := TRUE;
          "TI_PRESET_TEC_FLG" := 5;
       ELSE
          IF NOT "PDI".LS_TEC_FLG_DN THEN
             "PFM_TEC_FLG_DN"  := FALSE;
          END_IF;     
       END_IF;        

       // Lower furnace chamber swivel in [癩 


       "AV".LO_FCH_SW_ENC_POS := (DINT_TO_REAL(DWORD_TO_DINT("P_BM_LO_FCH_SW_ENC_POS":P))/#enc_inc_rot * "CNF".LO_FCH_SW_ENC_RATIO -90.0);   // 90,0=Offset encoder value
       #SET_REF_POS := DINT_TO_DWORD(REAL_TO_DINT(("CNF".LO_FCH_SW_REF_POS)/"CNF".LO_FCH_SW_ENC_RATIO* #enc_inc_rot));
       IF "DV".LO_FCH_SW_SET_REF_POS THEN
          "TI_PRESET_LO_FCH_SW" := "TI_PRESET_LO_FCH_SW" - 1;    
          "P_BM_LO_FCH_SW_ENC_REF":P := #SET_REF_POS OR 2#1000_0000_0000_0000_0000_0000_0000_0000;
       ELSE
          "P_BM_LO_FCH_SW_ENC_REF":P := #SET_REF_POS;
       END_IF;
       IF "PDI".LS_FCH_LFT_DN THEN
           "NFM_LS_FCH_LFT_DN" := TRUE;
       ELSE
          IF NOT "PDI".LS_FCH_LFT_DN AND "NFM_LS_FCH_LFT_DN" AND "PDI".LS_FCH_HOOK_WORK THEN
             "NFM_LS_FCH_LFT_DN" := FALSE;
             "TI_PRESET_LO_FCH_SW" := 3;     
          END_IF;
       END_IF;     
       "DV".LO_FCH_SW_SET_REF_POS := (("TI_PRESET_LO_FCH_SW" >0) AND ("TI_PRESET_LO_FCH_SW"<4)) OR "KYD".LO_FCH_SW_REF_SET;

       // Upper furnace chamber swivel in [癩  
       "AV".UP_FCH_SW_ENC_POS := (DINT_TO_REAL(DWORD_TO_DINT("P_BM_UP_FCH_SW_ENC_POS":P))/#enc_inc_rot *"CNF".UP_FCH_SW_ENC_RATIO)-90.0; // 90,0=Offset encoder value
       #SET_REF_POS := DINT_TO_DWORD(REAL_TO_DINT(("CNF".UP_FCH_SW_REF_POS)/"CNF".UP_FCH_SW_ENC_RATIO* #enc_inc_rot));
       IF "DV".UP_FCH_SW_SET_REF_POS THEN
          "TI_PRESET_UP_FCH_SW" := "TI_PRESET_UP_FCH_SW" - 1;
          "P_BM_UP_FCH_SW_ENC_REF":P := #SET_REF_POS OR 2#1000_0000_0000_0000_0000_0000_0000_0000;
       ELSE
          "P_BM_UP_FCH_SW_ENC_REF":P := 16#0000_0000;
       END_IF;

       "DV".UP_FCH_SW_SET_REF_POS :=  (("TI_PRESET_UP_FCH_SW" >0) AND ("TI_PRESET_UP_FCH_SW"<4)) OR "KYD".UP_FCH_SW_REF_SET;

